# EPICS alarm handler configuration: mps_database/bare/alarms/areas/mpln_sps_mp02.alhConfig
GROUP NULL MPLN:SPS:MP02:1
$ALIAS MPS Link Node 192
$GUIDANCE
LTUH MPS
   Group Name: MPLN:SPS:MP02:1
   Summary PV:  MPLN:SPS:MP02:1:STATSUMY
$END
CHANNEL  MPLN:SPS:MP02:1    MPLN:SPS:MP02:1:MPS_EN_RBV		-----
CHANNEL  MPLN:SPS:MP02:1    MPLN:SPS:MP02:1:LC1_MODE_RBV		-----
